PROGRAM PRG_TEST
VAR
	fbMotor_Test : FB_Motor_Test;
	fbTankTest : FB_TankTest;
END_VAR

TcUnit.RUN();

END_PROGRAM

(* stored: Version 1.1.0.1, ProductVersion 3.1.4024.16
   POU PRG_TEST: Id {9e50e3e8-5651-432a-a728-13b46bc2585b}, SpecialFunc None *)
